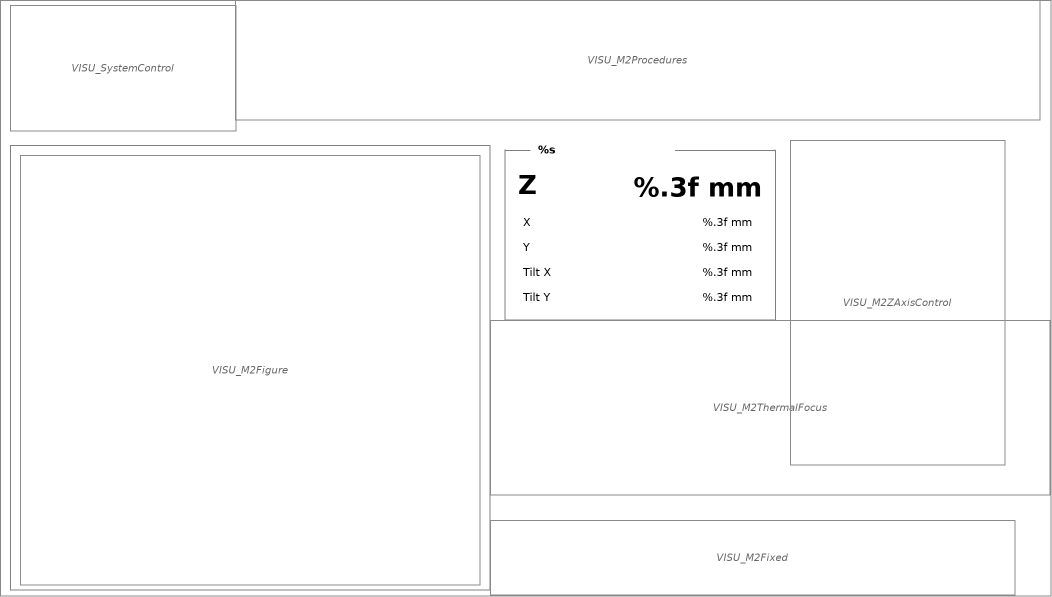
VISUALIZATION VISU_M2Overview  // 1052x597
VAR_IN_OUT
	ref : M2;
    widget : M2Widget;
END_VAR
    Polyline (675,150) (775,150) (775,320) (505,320) (505,150) (530,150)
    Rectangle (10,145 480x445)
    Frame (10,5 226x126)
        shows VISU_SystemControl(status := widget.actualStatus, button_initialize := widget.button_initialize, button_operating := widget.button_operating, button_locking := widget.button_locking)
    Frame (20,155 460x430)
        shows VISU_M2Figure(ref := ref, widget := widget.figure)
    Frame (235,0 805x120)
        shows VISU_M2Procedures(ref := ref, widget := widget)
    Rectangle (570,170 195x35), "%.3f mm", text variable: ref.parts.z.position.average.millimeters.value
        p55702900: widget.poweredColor
    Rectangle (650,210 105x25), "%.3f mm", text variable: ref.parts.x.position.average.millimeters.value
        p55702900: widget.poweredColor
    Rectangle (650,235 105x25), "%.3f mm", text variable: ref.parts.y.position.average.millimeters.value
        p55702900: widget.poweredColor
    Rectangle (650,285 105x25), "%.3f mm", text variable: ref.parts.tiltY.position.average.millimeters.value
        p55702900: widget.poweredColor
    Rectangle (650,260 105x25), "%.3f mm", text variable: ref.parts.tiltX.position.average.millimeters.value
        p55702900: widget.poweredColor
    Frame (490,320 560x175)
        shows VISU_M2ThermalFocus(ref := ref, widget := widget)
    Rectangle (535,135 150x30), "%s", text variable: widget.positionsTitle
    Rectangle (515,165 45x40), "Z"
        p55702900: widget.poweredColor
    Rectangle (520,210 45x25), "X"
        p55702900: widget.poweredColor
    Rectangle (520,235 45x25), "Y"
        p55702900: widget.poweredColor
    Rectangle (520,260 45x25), "Tilt X"
        p55702900: widget.poweredColor
    Rectangle (520,285 45x25), "Tilt Y"
        p55702900: widget.poweredColor
    Frame (790,140 215x325)
        shows VISU_M2ZAxisControl(widget := widget.z)
    Frame (490,520 525x75)
        shows VISU_M2Fixed(ref := ref, widget := widget)
END_VISUALIZATION

(* stored: Version 1.1.0.1, ProductVersion 3.1.4019.2
   Visu VISU_M2Overview: Id {16f3327f-b99c-49b2-b12d-b234eca9c341} *)
